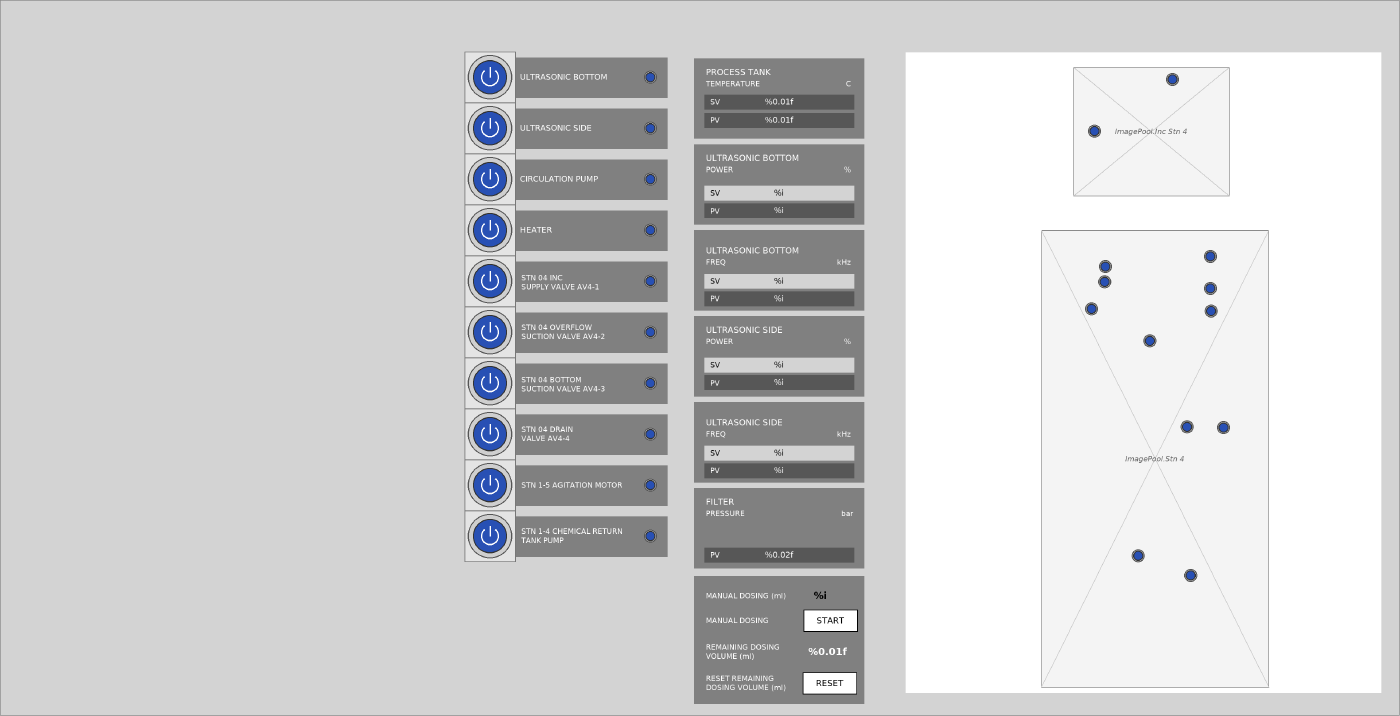
VISUALIZATION Manual_Station04  // 1920x983
    Rectangle (0,0 1920x983)
    Rectangle (1242,72 652x879)
    Image (1428,316 312x628), image: ImagePool.Stn 4
    RoundedRectangle (676,79 239x55)
    Label (710,98 163x16), "ULTRASONIC BOTTOM"
    Lamp1 (882,96 20x20), variable: ARdsMAP_HmiVariableStn[4].bProTankUsBtm_IND, style: Lamp-Lamp1-Blue
    PowerSwitch (637,71 70x70), variable: ARdsMAP_HmiVariableStn[4].bProTankUsBtm_PB, behaviour: TOGGLE, style: Switch-PowerSwitch-Blue
    RoundedRectangle (684,219 231x55)
    Label (710,238 151x16), "CIRCULATION PUMP"
    Lamp1 (882,236 20x20), variable: ARdsMAP_HmiVariableStn[4].bProTankPump_IND, style: Lamp-Lamp1-Blue
    PowerSwitch (637,211 70x70), variable: ARdsMAP_HmiVariableStn[4].bProTankPump_PB, behaviour: TOGGLE, style: Switch-PowerSwitch-Blue
    RoundedRectangle (684,289 231x55)
    Label (710,308 151x16), "HEATER"
    Lamp1 (882,306 20x20), variable: ARdsMAP_HmiVariableStn[4].bProTankHeater_IND, style: Lamp-Lamp1-Blue
    PowerSwitch (637,281 70x70), variable: ARdsMAP_HmiVariableStn[4].bProTankHeater_PB, behaviour: TOGGLE, style: Switch-PowerSwitch-Blue
    RoundedRectangle (676,149 239x55)
    Label (710,168 163x16), "ULTRASONIC SIDE"
    Lamp1 (882,166 20x20), variable: ARdsMAP_HmiVariableStn[4].bProTankUsSide_IND, style: Lamp-Lamp1-Blue
    PowerSwitch (637,141 70x70), variable: ARdsMAP_HmiVariableStn[4].bProTankUsSide_PB, behaviour: TOGGLE, style: Switch-PowerSwitch-Blue
    RoundedRectangle (684,429 231x55)
    Label (712,438 160x36), "STN 04 OVERFLOW SUCTION VALVE AV4-2"
    Lamp1 (882,446 20x20), variable: ARdsMAP_HmiVariableStn[4].bValve02_IND, style: Lamp-Lamp1-Blue
    PowerSwitch (637,421 70x70), variable: ARdsMAP_HmiVariableStn[4].bValve02_PB, behaviour: TOGGLE, style: Switch-PowerSwitch-Blue
    RoundedRectangle (684,359 231x55)
    Lamp1 (882,376 20x20), variable: ARdsMAP_HmiVariableStn[4].bValve01_IND, style: Lamp-Lamp1-Blue
    PowerSwitch (637,351 70x70), variable: ARdsMAP_HmiVariableStn[4].bValve01_PB, behaviour: TOGGLE, style: Switch-PowerSwitch-Blue
    Label (712,370 151x36), "STN 04 INC SUPPLY VALVE AV4-1"
    RoundedRectangle (684,569 231x55)
    Label (712,578 160x36), "STN 04 DRAIN VALVE AV4-4"
    Lamp1 (882,586 20x20), variable: ARdsMAP_HmiVariableStn[4].bValve04_IND, style: Lamp-Lamp1-Blue
    PowerSwitch (637,561 70x70), variable: ARdsMAP_HmiVariableStn[4].bValve04_PB, behaviour: TOGGLE, style: Switch-PowerSwitch-Blue
    RoundedRectangle (684,499 231x55)
    Lamp1 (882,516 20x20), variable: ARdsMAP_HmiVariableStn[4].bValve03_IND, style: Lamp-Lamp1-Blue
    PowerSwitch (637,491 70x70), variable: ARdsMAP_HmiVariableStn[4].bValve03_PB, behaviour: TOGGLE, style: Switch-PowerSwitch-Blue
    Label (712,510 151x36), "STN 04 BOTTOM SUCTION VALVE AV4-3"
    RoundedRectangle (684,639 231x55)
    Label (712,648 160x36), "STN 1-5 AGITATION MOTOR"
    Lamp1 (882,656 20x20), variable: ARdsMAP_HmiVariableGeneral.bProTankAgitationMotor_IND, style: Lamp-Lamp1-Blue
    PowerSwitch (637,631 70x70), variable: ARdsMAP_HmiVariableGeneral.bProTankAgitationMotor_PB, behaviour: TOGGLE, style: Switch-PowerSwitch-Blue
    RoundedRectangle (684,709 231x55)
    Label (712,718 160x36), "STN 1-4 CHEMICAL RETURN TANK PUMP"
    Lamp1 (882,726 20x20), variable: ARdsMAP_HmiVariableGeneral.bProTankPump_IND, style: Lamp-Lamp1-Blue
    PowerSwitch (637,701 70x70), variable: ARdsMAP_HmiVariableGeneral.bProTankPump_PB, behaviour: TOGGLE, style: Switch-PowerSwitch-Blue
    Lamp1 (1567,458 20x20), variable: ARdsMAP_HmiVariableStn[4].bProTankUsBtm_IND, style: Lamp-Lamp1-Blue
    Lamp1 (1551,753 20x20), variable: ARdsMAP_HmiVariableStn[4].bProTankPump_IND, style: Lamp-Lamp1-Blue
    Lamp1 (1505,377 20x20), variable: ARdsMAP_HmiVariableStn[4].bProTankHeater_IND, style: Lamp-Lamp1-Blue
    Lamp1 (1487,414 20x20), variable: ARdsMAP_HmiVariableStn[4].bProTankUsSide_IND, style: Lamp-Lamp1-Blue
    Lamp1 (1668,577 20x20), variable: ARdsMAP_HmiVariableStn[4].bValve02_IND, style: Lamp-Lamp1-Blue
    Lamp1 (1623,780 20x20), variable: ARdsMAP_HmiVariableStn[4].bValve04_IND, style: Lamp-Lamp1-Blue
    Lamp1 (1618,576 20x20), variable: ARdsMAP_HmiVariableStn[4].bValve03_IND, style: Lamp-Lamp1-Blue
    Lamp1 (1650,342 20x20), variable: ARdsMAP_HmiVariableStn[4].bOverflowMaxLevel_IND, style: Lamp-Lamp1-Blue
    Lamp1 (1506,356 20x20), variable: ARdsMAP_HmiVariableStn[4].bProcessTankMinLevel_IND, style: Lamp-Lamp1-Blue
    Lamp1 (1650,386 20x20), variable: ARdsMAP_HmiVariableStn[4].bOverflowMinLevel_IND, style: Lamp-Lamp1-Blue
    Lamp1 (1651,417 20x20), variable: ARdsMAP_HmiVariableStn[4].bProTankUsSide_IND, style: Lamp-Lamp1-Blue
    Image (1472,92 214x177), image: ImagePool.Inc Stn 4
    Lamp1 (1598,99 20x20), variable: ARdsMAP_HmiVariableStn[4].bValve01_IND, style: Lamp-Lamp1-Blue
    Lamp1 (1491,170 20x20), variable: ARdsMAP_HmiVariableStn[4].bDosingPump_IND, style: Lamp-Lamp1-Blue
    RoundedRectangle (952,791 233x175)
    Rectangle (1102,837 74x30), "START", colour toggle: ARbStnManualDosingST[4]
        toggle ARbStnManualDosingST[4]
    Label (965,838 109x28), "MANUAL DOSING"
    Label (965,804 121x28), "MANUAL DOSING (ml)"
    Rectangle (1084,804 82x28), "%i", text variable: ARDSProminentDosingHMI[4].In_iManualDosingVolume_ml
        OnMouseDown: write the text variable via VisuDialogs.Numpad, min 1, max 32767
    Label (965,924 129x28), "RESET REMAINING DOSING VOLUME (ml)"
    Rectangle (1101,923 74x30), "RESET", colour toggle: ARDSProminentDosingHMI[4].In_bResetRemainedDosingVolumePB
        tap ARDSProminentDosingHMI[1].In_bResetRemainedDosingVolumePB
    Label (965,881 118x28), "REMAINING DOSING VOLUME (ml)"
    Rectangle (1094,881 82x28), "%0.01f", text variable: ARDSProminentDosingHMI[4].Out_rRemainedDosingVolume_ml
    RoundedRectangle (952,80 233x110)
    Label (1141,104 29x22), "C"
    Rectangle (966,130 205x20), "%0.01f", text variable: ARrStnTempSV[4]
    Label (971,129 22x22), "SV"
    Rectangle (966,155 205x20), "%0.01f", text variable: ARrStnTempPV[4]
    Label (971,154 22x22), "PV"
    Label (965,91 150x16), "PROCESS TANK"
    Label (965,104 99x22), "TEMPERATURE"
    RoundedRectangle (952,198 233x110)
    Label (1141,222 29x22), "%"
    Rectangle (966,255 205x20), "%i", text variable: ARiStnManualUSBtmAsv[4]
        OnMouseDown: write the text variable via VisuDialogs.Numpad, min 10, max 100
    Label (971,254 22x22), "SV"
    Rectangle (966,279 205x20), "%i", text variable: ARiStnUSBtmAPv[4]
    Label (971,279 22x22), "PV"
    Label (965,209 150x16), "ULTRASONIC BOTTOM"
    Label (965,222 99x22), "POWER"
    RoundedRectangle (952,670 233x110)
    Label (1141,694 32x22), "bar"
    Rectangle (966,752 205x20), "%0.02f", text variable: ARrStnFilterPressurePV[4]
    Label (971,751 22x22), "PV"
    Label (965,681 150x16), "FILTER"
    Label (965,694 99x22), "PRESSURE"
    RoundedRectangle (952,316 233x110)
    Label (1141,349 29x22), "kHz"
    Rectangle (966,400 205x20), "%i", text variable: ARiStnUSBtmAFreqPv[4]
    Label (971,399 22x22), "PV"
    Rectangle (966,376 205x20), "%i", text variable: DSWeberEnclosure[2].DSWeberGenerator[1].DSWeberMulFreqSwitching.iFreqOutput_TS
        tap DSWeberEnclosure[2].DSWeberGenerator[1].DSWeberMulFreqSwitching.bFreqSwitchingPB_TS
    Label (971,375 22x22), "SV"
    Label (965,349 99x22), "FREQ"
    Label (965,336 150x16), "ULTRASONIC BOTTOM"
    RoundedRectangle (952,434 233x110)
    Label (1141,458 29x22), "%"
    Rectangle (966,491 205x20), "%i", text variable: ARiStnManualUSSideAsv[4]
        OnMouseDown: write the text variable via VisuDialogs.Numpad, min 10, max 100
    Label (971,490 22x22), "SV"
    Rectangle (966,515 205x20), "%i", text variable: ARiStnUSSideAPv[4]
    Label (971,515 22x22), "PV"
    Label (965,445 150x16), "ULTRASONIC SIDE"
    Label (965,458 99x22), "POWER"
    RoundedRectangle (952,552 233x110)
    Label (965,585 99x22), "FREQ"
    Label (965,572 150x16), "ULTRASONIC SIDE"
    Label (1141,585 29x22), "kHz"
    Rectangle (966,636 205x20), "%i", text variable: ARiStnUSSideAFreqPv[4]
    Label (971,635 22x22), "PV"
    Rectangle (966,612 205x20), "%i", text variable: DSWeberEnclosure[2].DSWeberGenerator[1].DSWeberMulFreqSwitching.iFreqOutput_TS
        tap DSWeberEnclosure[1].DSWeberGenerator[1].DSWeberMulFreqSwitching.bFreqSwitchingPB_TS
    Label (971,611 22x22), "SV"
END_VISUALIZATION

(* stored: Version 1.1.0.1, ProductVersion 3.1.4024.12
   Visu Manual_Station04: Id {cc4242fd-1208-4fb1-b41c-cf7f378edc55} *)
